TYPE ForceControlParam :
STRUCT

END_STRUCT
END_TYPE

(* stored: Version 1.1.0.1, ProductVersion 3.1.4024.11
   DUT ForceControlParam: Id {7df83d74-6eb0-4b15-98a4-abf6b02475da} *)
